Yaskawa INFORM job: 02-WORK_IN_STATION.JBI

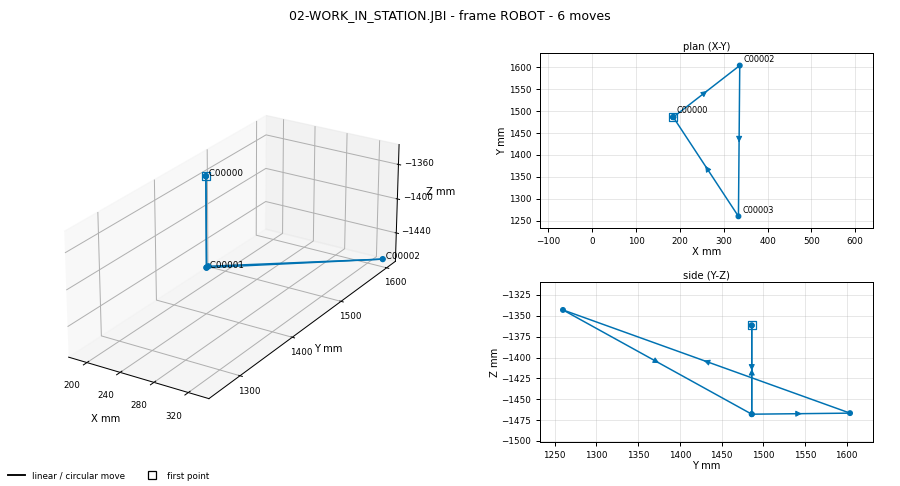
[picture p0: tool path of 02-WORK_IN_STATION.JBI in frame ROBOT, 6 of 6 moves have a stored position in this frame; points joined in program order, loops and branches not executed]
/JOB
//NAME 02-WORK_IN_STATION
///FOLDERNAME SAFETY
//POS
///NPOS 6,6,6,0,0,0
///TOOL 0
///POSTYPE ROBOT
///RECTAN
///RCONF 0,0,0,0,1,0,0,0,0,0,0,0,0,0,0,0,0,0,0,0,0,0,0,0
C00000=184.752,1486.138,-1361.526,-0.2468,-1.0938,97.3687
C00001=184.750,1486.139,-1467.927,-0.2465,-1.0940,97.3685
C00002=336.475,1603.929,-1466.658,-0.2065,-0.8510,132.5188
C00003=333.480,1259.846,-1342.970,13.7054,13.7763,133.9676
C00004=184.750,1486.139,-1467.927,-0.2465,-1.0940,97.3685
C00005=184.752,1486.138,-1361.526,-0.2468,-1.0938,97.3687
///RCONF 0,0,0,0,0,0,0,0,0,0,0,0,0,0,0,0,0,0,0,0,0,0,0,0
BC00000=1305.608,5117.603,449.998
BC00001=1305.608,5117.603,449.998
BC00002=1305.608,5117.603,449.998
BC00003=1305.608,5117.603,449.998
BC00004=1305.608,5117.603,449.998
BC00005=1305.608,5117.603,449.998
///POSTYPE PULSE
///PULSE
EC00000=0,-2782363
EC00001=0,-2782363
EC00002=0,-2565011
EC00003=-178256,-2565011
EC00004=0,-2782363
EC00005=0,-2782363
//INST
///DATE 2023/07/13 09:22
///ATTR SC,RW,RJ
////FRAME ROBOT
///GROUP1 RB1,BS1
///GROUP2 ST1
NOP
*START
MOVL C00000 BC00000 V=150.0  +MOVJ EC00000 VJ=100.00
MOVL C00001 BC00001 V=150.0  +MOVJ EC00001 VJ=100.00
SMOVL C00002 BC00002 V=150.0  +MOVJ EC00002
SMOVL C00003 BC00003 V=150.0  +MOVJ EC00003
SMOVL C00004 BC00004 V=150.0  +MOVJ EC00004
MOVL C00005 BC00005 V=150.0  +MOVJ EC00005 VJ=100.00
JUMP *START
END
